FUNCTION_BLOCK DoorControl
VAR_INPUT
END_VAR
VAR_OUTPUT
END_VAR
VAR
	r_doorTimer : TON;
END_VAR

//GVL_1.q_bOpenDoor := FALSE;
//GVL_1.q_bCloseDoor := FALSE;

IF GVL_1.i_iCurrentFloor = GVL_1.g_iTargetFloor THEN
    GVL_1.q_bOpenDoor := TRUE;
	GVL_1.q_bCloseDoor := FALSE;
    r_doorTimer(IN := TRUE, PT := T#10S);
ELSE
    GVL_1.q_bCloseDoor := TRUE;
	GVL_1.q_bOpenDoor := FALSE;
    r_doorTimer(IN := FALSE);
END_IF

IF r_doorTimer.Q THEN
    GVL_1.q_bOpenDoor := FALSE;
    GVL_1.q_bCloseDoor := TRUE;
	r_doorTimer(IN := FALSE);
END_IF

END_FUNCTION_BLOCK

(* stored: Version 1.1.0.1, ProductVersion 3.1.4024.15
   POU DoorControl: Id {7e541a19-8749-4c57-8e90-e24ffb0f778c}, SpecialFunc None *)
